{attribute 'GeneratedUsingTerminal: EL3773-0000-0021'}
{attribute addProperty BoxType "EL3773-0000-0021"}
{attribute addProperty Id "U2_SamplesAT %I*U2_Samples_2549228720"}
{attribute addProperty CRC "1977103279"}
{attribute addProperty Size "20"}
TYPE L2_Voltage_Samples_75D833AF EXTENDS TcoIo.InputBase_8311D824 :
STRUCT
	{attribute addProperty Name "U2_Samples"}
	U2_Samples AT %I* : U2_Samples_25492287;
END_STRUCT
END_TYPE

(* stored: Version 1.2.0.0, ProductVersion 3.1.4024.11
   DUT L2_Voltage_Samples_75D833AF: Id {c7bc6ce7-b05e-007b-1382-1ccd736c69dc} *)
